FUNCTION_BLOCK splitCameraInfo (* Tamplate for a simple Basic Function Block Type *)
  (* Standard: 61499-2 *)
  (* Version 0.0, 2018-01-23, 4DIAC-IDE, 4DIAC-Consortium *)
  (* Version 1.0, 2016-05-26, AZ, fortiss GmbH *)
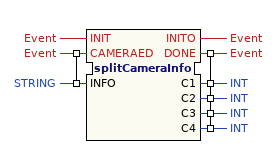
  EVENT_INPUT
    INIT; (* Initialization Request *)
    CAMERAED WITH INFO; (* Normal Execution Request *)
  END_EVENT
  EVENT_OUTPUT
    INITO; (* Initialization Confirm *)
    DONE WITH C1, C2, C3, C4; (* Execution Confirmation *)
  END_EVENT
  VAR_INPUT
    INFO : STRING; (* Input event qualifier *)
  END_VAR
  VAR_OUTPUT
    C1 : INT;
    C2 : INT;
    C3 : INT;
    C4 : INT;
  END_VAR
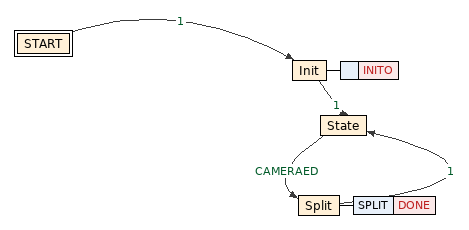
  EC_STATES
    START; (* Initial State *)
    Init : -> INITO; (* Initialization *)
    Split : SPLIT -> DONE;
    State;
  END_STATES
  EC_TRANSITIONS
    START TO Init := 1;
    Split TO State := 1;
    State TO Split := CAMERAED;
    Init TO State := 1;
  END_TRANSITIONS
  ALGORITHM SPLIT IN ST: (* new algorithm *)

  END_ALGORITHM
END_FUNCTION_BLOCK
